{attribute 'qualified_only'}
{attribute 'strict'}
TYPE eDelayType :
(
	Immediate := 0,
	DelayByTimer := 1,
	DelayByPos := 2
);
END_TYPE

(* stored: Version 1.1.0.1, ProductVersion 3.1.4024.3
   EnumerationTextList eDelayType: Id {43257eb7-31c4-0073-2afe-1c889abebd0c} *)
